FUNCTION_BLOCK UDINT_Array
VAR_GENERIC CONSTANT
	MX		: UDINT := 1;
	MI		: UDINT := 1;
END_VAR
VAR
	_nArray	: ARRAY[MI..MX] OF UDINT;
	_nHead	: UDINT;
	_nTail	: UDINT;
END_VAR

METHOD Get : Results.Result
VAR_INPUT
	nPos		: UDINT;
END_VAR
VAR_OUTPUT
	nVal		: UDINT;
END_VAR
IF nPos < MI OR nPos > MX THEN
	Get := Results.Error;
	RETURN;
END_IF


nVal := _nArray[nPos];
Get := Results.Ok;
END_METHOD

METHOD Pop : Results.Result
VAR_OUTPUT
    nVal    : UDINT;
END_VAR
IF _nHead = _nTail THEN
    Pop := Results.Error;
    RETURN;
END_IF

nVal := _nArray[_nTail];

_nTail := (_nTail + 1) MOD (MX - MI + 1);

Pop := Results.Ok;
END_METHOD

METHOD Push : Results.Result
VAR_INPUT
    nVal    : UDINT;
END_VAR
IF (_nHead + 1) MOD (MX - MI + 1) = _nTail THEN
    Push := Results.Error;
    RETURN;
END_IF

_nArray[_nHead] := nVal;

_nHead := (_nHead + 1) MOD (MX - MI + 1);

Push := Results.Ok;
END_METHOD

METHOD Set : UDINT
VAR_INPUT
	nPos		: UDINT;
	nVal		: UDINT;
END_VAR
IF nPos < MI OR nPos > MX THEN
	Get := Results.Error;
	RETURN;
END_IF


_nArray[nPos] := nVal;
Get := Results.Ok;
END_METHOD

END_FUNCTION_BLOCK

(* stored: Version 1.1.0.1
   POU UDINT_Array: Id {6beeae34-1876-4583-b54c-fec934e67283}, SpecialFunc None
   Method Get: Id {50d45214-fc7c-468e-bc96-136d66d8d035}
   Method Pop: Id {9dafa2b2-c4d9-405e-ae03-7b86841e57aa}
   Method Push: Id {014e7f24-2205-43b5-a008-1708c183fb13}
   Method Set: Id {e272d147-4fee-4862-90da-40e1ad50f7a4} *)
